FUNCTION_BLOCK SUB_3_TEST (* Test SUB_3_LLP in a Composite Function Block *)
  (* Standard: 61499-2 *)
  (* Version 0.0, 2002-12-17, JHC, Rockwell Automation *)
  (* Compiler header: package fb.rt.test; *)
  (* Compiler Java IBM Jikes 1.06 *)
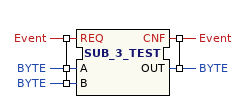
  EVENT_INPUT
    REQ WITH A, B; (* Normal Execution Request *)
  END_EVENT
  EVENT_OUTPUT
    CNF WITH OUT; (* Execution Confirmation *)
  END_EVENT
  VAR_INPUT
    A : BYTE;
    B : BYTE;
  END_VAR
  VAR_OUTPUT
    OUT : BYTE; (* Output event qualifier *)
  END_VAR
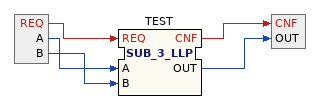
  FBS
    TEST : SUB_3_LLP;
  END_FBS
  EVENT_CONNECTIONS
    REQ TO TEST.REQ;
    TEST.CNF TO CNF;
  END_CONNECTIONS
  DATA_CONNECTIONS
    A TO TEST.A;
    B TO TEST.B;
    TEST.OUT TO OUT;
  END_CONNECTIONS
END_FUNCTION_BLOCK
